FUNCTION_BLOCK FB_Zentral_TaktimpulsGenerator
VAR_INPUT
	Ir_Frequenz		: REAL; 
END_VAR
VAR_OUTPUT
	Ox_Takt								: BOOL; 
	Ox_Impuls							: BOOL; 
END_VAR

VAR
	St_TakttimerEinfach					: TON; 
	ReadRTC									: R_SYS_T; 
	TimeValid									: BOOL; 
	RTCTime									: DT; 
	RTCMillis									: DWORD; 
	Sdt_StartAktuellerTakt				: DT; 
	Sx_TaktFP								: BOOL; 
	Sx_Init										: BOOL; 
	St_DifferenzStartAktuell			:TIME; 	
	Sdw_StartAktuellerTaktMillis	:DWORD;  
END_VAR
	
VAR_TEMP

END_VAR

//Erfassung aktuelle Date and Time
ReadRTC(It_SynchTime := T#5S, Ox_TimeValid => TimeValid, Odt_RTCTime => RTCTime, Odw_Milliseconds => RTCMillis);  
	
//Ermittlung Dauer seit Taktstart
St_DifferenzStartAktuell := T_DIFF(Idt_Time1 := RTCTime, Idw_Time1Millis :=RTCMillis, Idt_Time2 := Sdt_StartAktuellerTakt, Idw_Time2Millis := Sdw_StartAktuellerTaktMillis); 


//Taktbildung (halbe Zeit an/ halbe Zeit aus)
Ox_Takt := St_DifferenzStartAktuell > DINT_TO_TIME(REAL_TO_DINT((1000/Ir_Frequenz)/2)); 
	
//Impuls Takt 
Ox_Impuls := Ox_Takt AND NOT Sx_TaktFP;
Sx_TaktFP := Ox_Takt; 
	
//Abspeichern Start aktueller Takt
IF (St_DifferenzStartAktuell > DINT_TO_TIME(REAL_TO_DINT((1000/Ir_Frequenz)))) OR NOT Sx_Init THEN 
	Sdt_StartAktuellerTakt := RTCTime; 
	Sdw_StartAktuellerTaktMillis := RTCMillis; 
END_IF
	
//Baustein als initialisiert setzen 
Sx_Init := TRUE;

END_FUNCTION_BLOCK

(* stored: Version 1.1.0.1, ProductVersion 3.1.4024.9
   POU FB_Zentral_TaktimpulsGenerator: Id {817bfbbb-4fef-4ec8-9fa6-ce1ce00e14fc}, SpecialFunc None *)
